// TIA Portal V16 export
// export: Created 2021-11-12T13:33:06.2135503Z, ExportSetting WithDefaults, DisplayName Totally Integrated Automation Portal, DisplayVersion V16 Update 3, DisplayName TIA Portal Version Control Interface, DisplayVersion V16 Update 2, DisplayName TIA Portal Openness, DisplayVersion V16 Update 3, DisplayName SINAMICS Startdrive Advanced, DisplayVersion V16 Update 5, DisplayName SINAMICS Startdrive G130, G150, S120, S150, SINAMICS MV, S210, DisplayVersion V16 Update 5, DisplayName SINAMICS Startdrive G110M, G120, G120C, G120D, G120P, G115D, DisplayVersion V16 Update 5, DisplayName STEP 7 Professional, DisplayVersion V16 Update 3, DisplayName STEP 7 Safety, DisplayVersion V16, DisplayName WinCC UA Professional, DisplayVersion V16 Update 3
FUNCTION_BLOCK "IM_410+UH31+KF10"   // FB52, LAD
{ S7_Optimized_Access := 'TRUE' }
VERSION : 0.1
// stored: AutoNumber true, IsIECCheckEnabled false, IsRetainMemResEnabled false, MemoryReserve 100, SetENOAutomatically false, UDAEnableTagReadback false
   VAR
      KF11_Ix0 : "STD_CH_DI";
      KF11_Ix1 { S7_SetPoint := 'True'} : "STD_CH_DI";
      KF11_Ix2 { S7_SetPoint := 'True'} : "STD_CH_DI";
      KF11_Ix3 { S7_SetPoint := 'True'} : "STD_CH_DI";
      KF11_Ix4 { S7_SetPoint := 'True'} : "STD_CH_DI";
      KF11_Ix5 { S7_SetPoint := 'True'} : "STD_CH_DI";
      KF11_Ix6 { S7_SetPoint := 'True'} : "STD_CH_DI";
      KF11_Ix7 { S7_SetPoint := 'True'} : "STD_CH_DI";
      KF12_Ix0 { S7_SetPoint := 'True'} : "STD_CH_DI";
      KF12_Ix1 { S7_SetPoint := 'True'} : "STD_CH_DI";
      KF12_Ix2 { S7_SetPoint := 'True'} : "STD_CH_DI";
      KF12_Ix3 { S7_SetPoint := 'True'} : "STD_CH_DI";
      KF12_Ix4 { S7_SetPoint := 'True'} : "STD_CH_DI";
      KF12_Ix5 { S7_SetPoint := 'True'} : "STD_CH_DI";
      KF12_Ix6 { S7_SetPoint := 'True'} : "STD_CH_DI";
      KF12_Ix7 { S7_SetPoint := 'True'} : "STD_CH_DI";
      KF51_AI0 { S7_SetPoint := 'True'} : "STD_CH_AI";
      KF51_AI1 { S7_SetPoint := 'True'} : "STD_CH_AI";
      KF52_AI0 { S7_SetPoint := 'True'} : "STD_CH_AI";
      KF52_AI1 { S7_SetPoint := 'True'} : "STD_CH_AI";
   END_VAR
   VAR_TEMP   // added for the SCL form of the ladder/FBD networks
      _w1 : Bool;
      _w2 : Bool;
      _w3 : Bool;
   END_VAR
BEGIN

REGION Network 1: Module position -KF11
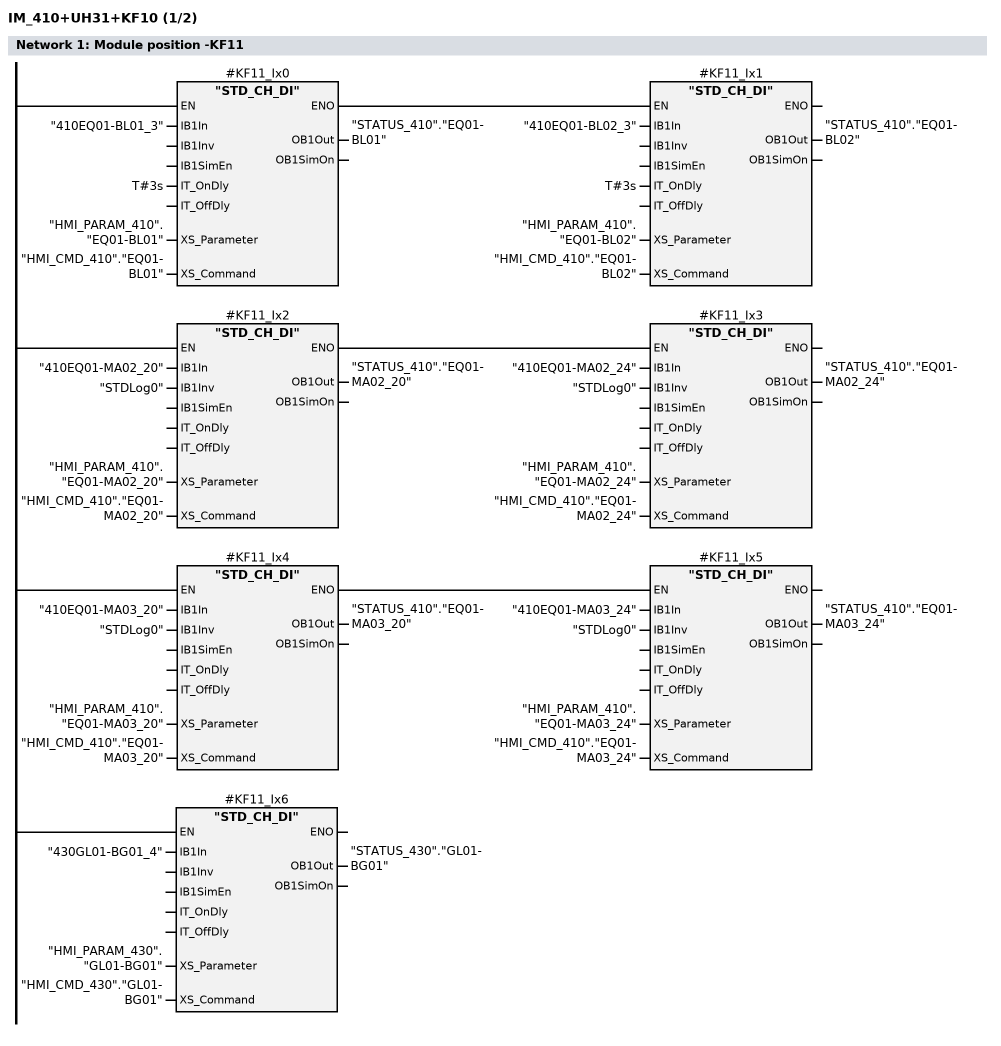
   RUNG wire#powerrail
      #KF11_Ix0(IB1In := "410EQ01-BL01_3", IB1Inv :=, IB1SimEn :=, IT_OnDly := T#3s, IT_OffDly :=, XS_Parameter := "HMI_PARAM_410"."EQ01-BL01", XS_Command := "HMI_CMD_410"."EQ01-BL01", OB1Out => "STATUS_410"."EQ01-BL01", OB1SimOn =>)
      #KF11_Ix1(IB1In := "410EQ01-BL02_3", IB1Inv :=, IB1SimEn :=, IT_OnDly := T#3s, IT_OffDly :=, XS_Parameter := "HMI_PARAM_410"."EQ01-BL02", XS_Command := "HMI_CMD_410"."EQ01-BL02", OB1Out => "STATUS_410"."EQ01-BL02", OB1SimOn =>)
   END_RUNG
   RUNG wire#powerrail
      #KF11_Ix2(IB1In := "410EQ01-MA02_20", IB1Inv := "STDLog0", IB1SimEn :=, IT_OnDly :=, IT_OffDly :=, XS_Parameter := "HMI_PARAM_410"."EQ01-MA02_20", XS_Command := "HMI_CMD_410"."EQ01-MA02_20", OB1Out => "STATUS_410"."EQ01-MA02_20", OB1SimOn =>)
      #KF11_Ix3(IB1In := "410EQ01-MA02_24", IB1Inv := "STDLog0", IB1SimEn :=, IT_OnDly :=, IT_OffDly :=, XS_Parameter := "HMI_PARAM_410"."EQ01-MA02_24", XS_Command := "HMI_CMD_410"."EQ01-MA02_24", OB1Out => "STATUS_410"."EQ01-MA02_24", OB1SimOn =>)
   END_RUNG
   RUNG wire#powerrail
      #KF11_Ix4(IB1In := "410EQ01-MA03_20", IB1Inv := "STDLog0", IB1SimEn :=, IT_OnDly :=, IT_OffDly :=, XS_Parameter := "HMI_PARAM_410"."EQ01-MA03_20", XS_Command := "HMI_CMD_410"."EQ01-MA03_20", OB1Out => "STATUS_410"."EQ01-MA03_20", OB1SimOn =>)
      #KF11_Ix5(IB1In := "410EQ01-MA03_24", IB1Inv := "STDLog0", IB1SimEn :=, IT_OnDly :=, IT_OffDly :=, XS_Parameter := "HMI_PARAM_410"."EQ01-MA03_24", XS_Command := "HMI_CMD_410"."EQ01-MA03_24", OB1Out => "STATUS_410"."EQ01-MA03_24", OB1SimOn =>)
   END_RUNG
   RUNG wire#powerrail
      #KF11_Ix6(IB1In := "430GL01-BG01_4", IB1Inv :=, IB1SimEn :=, IT_OnDly :=, IT_OffDly :=, XS_Parameter := "HMI_PARAM_430"."GL01-BG01", XS_Command := "HMI_CMD_430"."GL01-BG01", OB1Out => "STATUS_430"."GL01-BG01", OB1SimOn =>)
   END_RUNG
   // the same network as SCL:
   #KF11_Ix0(IB1In := "410EQ01-BL01_3",   // "STD_CH_DI"
             IT_OnDly := T#3s,
             XS_Parameter := "HMI_PARAM_410"."EQ01-BL01",
             XS_Command := "HMI_CMD_410"."EQ01-BL01",
             OB1Out => "STATUS_410"."EQ01-BL01",
             ENO => #_w1);
   IF #_w1 THEN
       #KF11_Ix1(IB1In := "410EQ01-BL02_3",   // "STD_CH_DI"
                 IT_OnDly := T#3s,
                 XS_Parameter := "HMI_PARAM_410"."EQ01-BL02",
                 XS_Command := "HMI_CMD_410"."EQ01-BL02",
                 OB1Out => "STATUS_410"."EQ01-BL02");
   END_IF;
   #KF11_Ix2(IB1In := "410EQ01-MA02_20",   // "STD_CH_DI"
             IB1Inv := "STDLog0",
             XS_Parameter := "HMI_PARAM_410"."EQ01-MA02_20",
             XS_Command := "HMI_CMD_410"."EQ01-MA02_20",
             OB1Out => "STATUS_410"."EQ01-MA02_20",
             ENO => #_w2);
   IF #_w2 THEN
       #KF11_Ix3(IB1In := "410EQ01-MA02_24",   // "STD_CH_DI"
                 IB1Inv := "STDLog0",
                 XS_Parameter := "HMI_PARAM_410"."EQ01-MA02_24",
                 XS_Command := "HMI_CMD_410"."EQ01-MA02_24",
                 OB1Out => "STATUS_410"."EQ01-MA02_24");
   END_IF;
   #KF11_Ix4(IB1In := "410EQ01-MA03_20",   // "STD_CH_DI"
             IB1Inv := "STDLog0",
             XS_Parameter := "HMI_PARAM_410"."EQ01-MA03_20",
             XS_Command := "HMI_CMD_410"."EQ01-MA03_20",
             OB1Out => "STATUS_410"."EQ01-MA03_20",
             ENO => #_w3);
   IF #_w3 THEN
       #KF11_Ix5(IB1In := "410EQ01-MA03_24",   // "STD_CH_DI"
                 IB1Inv := "STDLog0",
                 XS_Parameter := "HMI_PARAM_410"."EQ01-MA03_24",
                 XS_Command := "HMI_CMD_410"."EQ01-MA03_24",
                 OB1Out => "STATUS_410"."EQ01-MA03_24");
   END_IF;
   #KF11_Ix6(IB1In := "430GL01-BG01_4",   // "STD_CH_DI"
             XS_Parameter := "HMI_PARAM_430"."GL01-BG01",
             XS_Command := "HMI_CMD_430"."GL01-BG01",
             OB1Out => "STATUS_430"."GL01-BG01");
END_REGION

REGION Network 2: Module position -KF12
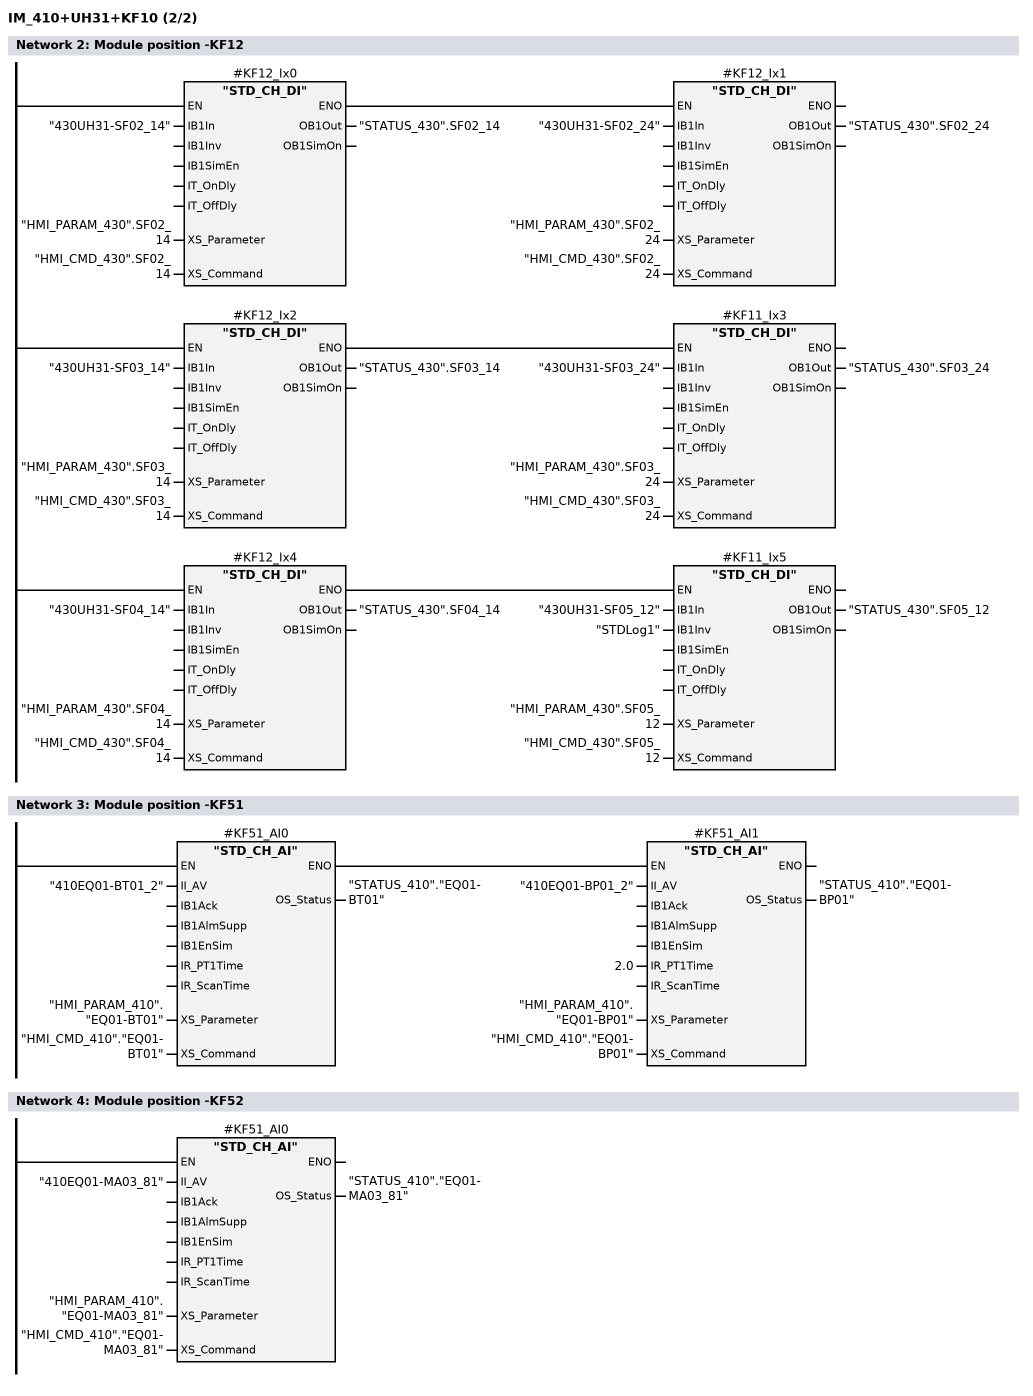
   RUNG wire#powerrail
      #KF12_Ix0(IB1In := "430UH31-SF02_14", IB1Inv :=, IB1SimEn :=, IT_OnDly :=, IT_OffDly :=, XS_Parameter := "HMI_PARAM_430".SF02_14, XS_Command := "HMI_CMD_430".SF02_14, OB1Out => "STATUS_430".SF02_14, OB1SimOn =>)
      #KF12_Ix1(IB1In := "430UH31-SF02_24", IB1Inv :=, IB1SimEn :=, IT_OnDly :=, IT_OffDly :=, XS_Parameter := "HMI_PARAM_430".SF02_24, XS_Command := "HMI_CMD_430".SF02_24, OB1Out => "STATUS_430".SF02_24, OB1SimOn =>)
   END_RUNG
   RUNG wire#powerrail
      #KF12_Ix2(IB1In := "430UH31-SF03_14", IB1Inv :=, IB1SimEn :=, IT_OnDly :=, IT_OffDly :=, XS_Parameter := "HMI_PARAM_430".SF03_14, XS_Command := "HMI_CMD_430".SF03_14, OB1Out => "STATUS_430".SF03_14, OB1SimOn =>)
      #KF11_Ix3(IB1In := "430UH31-SF03_24", IB1Inv :=, IB1SimEn :=, IT_OnDly :=, IT_OffDly :=, XS_Parameter := "HMI_PARAM_430".SF03_24, XS_Command := "HMI_CMD_430".SF03_24, OB1Out => "STATUS_430".SF03_24, OB1SimOn =>)
   END_RUNG
   RUNG wire#powerrail
      #KF12_Ix4(IB1In := "430UH31-SF04_14", IB1Inv :=, IB1SimEn :=, IT_OnDly :=, IT_OffDly :=, XS_Parameter := "HMI_PARAM_430".SF04_14, XS_Command := "HMI_CMD_430".SF04_14, OB1Out => "STATUS_430".SF04_14, OB1SimOn =>)
      #KF11_Ix5(IB1In := "430UH31-SF05_12", IB1Inv := "STDLog1", IB1SimEn :=, IT_OnDly :=, IT_OffDly :=, XS_Parameter := "HMI_PARAM_430".SF05_12, XS_Command := "HMI_CMD_430".SF05_12, OB1Out => "STATUS_430".SF05_12, OB1SimOn =>)
   END_RUNG
   // the same network as SCL:
   #KF12_Ix0(IB1In := "430UH31-SF02_14",   // "STD_CH_DI"
             XS_Parameter := "HMI_PARAM_430".SF02_14,
             XS_Command := "HMI_CMD_430".SF02_14,
             OB1Out => "STATUS_430".SF02_14,
             ENO => #_w1);
   IF #_w1 THEN
       #KF12_Ix1(IB1In := "430UH31-SF02_24",   // "STD_CH_DI"
                 XS_Parameter := "HMI_PARAM_430".SF02_24,
                 XS_Command := "HMI_CMD_430".SF02_24,
                 OB1Out => "STATUS_430".SF02_24);
   END_IF;
   #KF12_Ix2(IB1In := "430UH31-SF03_14",   // "STD_CH_DI"
             XS_Parameter := "HMI_PARAM_430".SF03_14,
             XS_Command := "HMI_CMD_430".SF03_14,
             OB1Out => "STATUS_430".SF03_14,
             ENO => #_w2);
   IF #_w2 THEN
       #KF11_Ix3(IB1In := "430UH31-SF03_24",   // "STD_CH_DI"
                 XS_Parameter := "HMI_PARAM_430".SF03_24,
                 XS_Command := "HMI_CMD_430".SF03_24,
                 OB1Out => "STATUS_430".SF03_24);
   END_IF;
   #KF12_Ix4(IB1In := "430UH31-SF04_14",   // "STD_CH_DI"
             XS_Parameter := "HMI_PARAM_430".SF04_14,
             XS_Command := "HMI_CMD_430".SF04_14,
             OB1Out => "STATUS_430".SF04_14,
             ENO => #_w3);
   IF #_w3 THEN
       #KF11_Ix5(IB1In := "430UH31-SF05_12",   // "STD_CH_DI"
                 IB1Inv := "STDLog1",
                 XS_Parameter := "HMI_PARAM_430".SF05_12,
                 XS_Command := "HMI_CMD_430".SF05_12,
                 OB1Out => "STATUS_430".SF05_12);
   END_IF;
END_REGION

REGION Network 3: Module position -KF51
   RUNG wire#powerrail
      #KF51_AI0(II_AV := "410EQ01-BT01_2", IB1Ack :=, IB1AlmSupp :=, IB1EnSim :=, IR_PT1Time :=, IR_ScanTime :=, XS_Parameter := "HMI_PARAM_410"."EQ01-BT01", XS_Command := "HMI_CMD_410"."EQ01-BT01", OS_Status => "STATUS_410"."EQ01-BT01")
      #KF51_AI1(II_AV := "410EQ01-BP01_2", IB1Ack :=, IB1AlmSupp :=, IB1EnSim :=, IR_PT1Time := 2.0, IR_ScanTime :=, XS_Parameter := "HMI_PARAM_410"."EQ01-BP01", XS_Command := "HMI_CMD_410"."EQ01-BP01", OS_Status => "STATUS_410"."EQ01-BP01")
   END_RUNG
   // the same network as SCL:
   #KF51_AI0(II_AV := "410EQ01-BT01_2",   // "STD_CH_AI"
             XS_Parameter := "HMI_PARAM_410"."EQ01-BT01",
             XS_Command := "HMI_CMD_410"."EQ01-BT01",
             OS_Status => "STATUS_410"."EQ01-BT01",
             ENO => #_w1);
   IF #_w1 THEN
       #KF51_AI1(II_AV := "410EQ01-BP01_2",   // "STD_CH_AI"
                 IR_PT1Time := 2.0,
                 XS_Parameter := "HMI_PARAM_410"."EQ01-BP01",
                 XS_Command := "HMI_CMD_410"."EQ01-BP01",
                 OS_Status => "STATUS_410"."EQ01-BP01");
   END_IF;
END_REGION

REGION Network 4: Module position -KF52
   RUNG wire#powerrail
      #KF51_AI0(II_AV := "410EQ01-MA03_81", IB1Ack :=, IB1AlmSupp :=, IB1EnSim :=, IR_PT1Time :=, IR_ScanTime :=, XS_Parameter := "HMI_PARAM_410"."EQ01-MA03_81", XS_Command := "HMI_CMD_410"."EQ01-MA03_81", OS_Status => "STATUS_410"."EQ01-MA03_81")
   END_RUNG
   // the same network as SCL:
   #KF51_AI0(II_AV := "410EQ01-MA03_81",   // "STD_CH_AI"
             XS_Parameter := "HMI_PARAM_410"."EQ01-MA03_81",
             XS_Command := "HMI_CMD_410"."EQ01-MA03_81",
             OS_Status => "STATUS_410"."EQ01-MA03_81");
END_REGION
END_FUNCTION_BLOCK
